// Test-only concrete child of FB_DeviceBase. Exposes the protected API
// (_Raise / _ClearFault / _AcceptCommand / _UpdateHeader) through public
// "Probe*" wrappers so FB_DeviceBase_Test can drive the base contract
// without a full device FB in the way. Also overrides ResolveFaultString
// so the tests can verify virtual dispatch.
//
// This FB lives in the Testing project on purpose — it is not part of the
// TcForge public surface.
FUNCTION_BLOCK FB_DeviceBase_Probe EXTENDS TcForge.FB_DeviceBase
VAR_OUTPUT
    header : TcForge.ST_DeviceHeader_Sts;
END_VAR

// Nothing cyclic — tests call the probe methods directly.

METHOD PUBLIC ProbeRaise : BOOL
VAR_INPUT
    code   : DINT;
    source : STRING(31);
    reason : STRING(79);
END_VAR
ProbeRaise := _Raise(code := code, source := source, reason := reason);
END_METHOD

METHOD PUBLIC ProbeClearFault
_ClearFault();
END_METHOD

METHOD PUBLIC ProbeAcceptCommand
VAR_INPUT
    eRequester : TcForge.E_Requester;
END_VAR
_AcceptCommand(eRequester := eRequester);
END_METHOD

// Populate the probe's own header struct via the protected _UpdateHeader.
METHOD PUBLIC Refresh
VAR_INPUT
    stateString : STRING(31);
    stsBusy     : BOOL;
END_VAR
_UpdateHeader(
    header      := header,
    stateString := stateString,
    stsBusy     := stsBusy);
END_METHOD

// Minimal resolver so the tests can verify virtual dispatch through the
// base's GetFaultString() / _UpdateHeader() calls. Maps a few well-known
// codes; everything else returns empty (inherited default behaviour).
METHOD PROTECTED ResolveFaultString : STRING(79)
VAR_INPUT
    code : DINT;
END_VAR
CASE code OF
    42: ResolveFaultString := 'Motion timeout';
    99: ResolveFaultString := 'Limit tripped';
ELSE
    ResolveFaultString := '';
END_CASE;
END_METHOD

END_FUNCTION_BLOCK

(* stored: Version 1.1.0.1, ProductVersion 3.1.4026.12
   POU FB_DeviceBase_Probe: Id {b1c2d3e4-f5a6-7890-abcd-000000000500}, SpecialFunc None
   Method ProbeRaise: Id {b1c2d3e4-f5a6-7890-abcd-000000000501}
   Method ProbeClearFault: Id {b1c2d3e4-f5a6-7890-abcd-000000000502}
   Method ProbeAcceptCommand: Id {b1c2d3e4-f5a6-7890-abcd-000000000503}
   Method Refresh: Id {b1c2d3e4-f5a6-7890-abcd-000000000504}
   Method ResolveFaultString: Id {b1c2d3e4-f5a6-7890-abcd-000000000505} *)
